{attribute 'GeneratedUsingTerminal: EK1122-0000-0018'}
{attribute addProperty BoxType "EK1122-0000-0018"}
{attribute addProperty Id "Beckhoff_EK15xxsub_EK1100EK1100_AB5A94672A_0001_EK1501_0000_0016EK1501_C99C274C6A_0002_EK1501_0000_0017EK1501_C99C274C6A_0003_EK1501_0000_0018EK1501_C99C274C6A_0004_EK1501_0000_0019EK1501_C99C274C6A_0005_EK1501_0010_0016EK1501_C99C274C6A_0006_EK1501_0010_0017EK1501_C99C274C6A_0007_EK1501_0010_0018EK1501_C99C274C6A_0008_EK1501_0100_0016EK1501_C99C274C6A_0020_EK1541_0000_0016EK1541_C99C274C6A_0021_EK1541_0000_0017EK1541_C99C274C6A_0022_EK1541_0000_0018EK1541_C99C274C6"}
{attribute addProperty CRC "2792001901"}
{attribute addProperty Size "68"}
TYPE Beckhoff_EK15xxEK1122_A66A916D EXTENDS EK1122_AB5A9467 :
STRUCT
	{attribute addProperty Name "Beckhoff_EK15xxsub_EK1100"}
	Beckhoff_EK15xxsub_EK1100 : EK1100_AB5A9467;
	{attribute addProperty Name "A_0001_EK1501_0000_0016"}
	A_0001_EK1501_0000_0016 : EK1501_C99C274C;
	{attribute addProperty Name "A_0002_EK1501_0000_0017"}
	A_0002_EK1501_0000_0017 : EK1501_C99C274C;
	{attribute addProperty Name "A_0003_EK1501_0000_0018"}
	A_0003_EK1501_0000_0018 : EK1501_C99C274C;
	{attribute addProperty Name "A_0004_EK1501_0000_0019"}
	A_0004_EK1501_0000_0019 : EK1501_C99C274C;
	{attribute addProperty Name "A_0005_EK1501_0010_0016"}
	A_0005_EK1501_0010_0016 : EK1501_C99C274C;
	{attribute addProperty Name "A_0006_EK1501_0010_0017"}
	A_0006_EK1501_0010_0017 : EK1501_C99C274C;
	{attribute addProperty Name "A_0007_EK1501_0010_0018"}
	A_0007_EK1501_0010_0018 : EK1501_C99C274C;
	{attribute addProperty Name "A_0008_EK1501_0100_0016"}
	A_0008_EK1501_0100_0016 : EK1501_C99C274C;
	{attribute addProperty Name "A_0020_EK1541_0000_0016"}
	A_0020_EK1541_0000_0016 : EK1541_C99C274C;
	{attribute addProperty Name "A_0021_EK1541_0000_0017"}
	A_0021_EK1541_0000_0017 : EK1541_C99C274C;
	{attribute addProperty Name "A_0022_EK1541_0000_0018"}
	A_0022_EK1541_0000_0018 : EK1541_C99C274C;
END_STRUCT
END_TYPE

(* stored: Version 1.2.0.0, ProductVersion 3.1.4024.9
   DUT Beckhoff_EK15xxEK1122_A66A916D: Id {f7227222-804a-4026-963d-04bd36e6b6af} *)
